// TIA Portal project "deneme3" (V14)

(* hardware
DEVICE "HMI_1"  KTP600 Basic color PN
   slot 0: "KTP600 Basic color PN"  KTP600 Basic color PN  6AV6 647-0AD11-3AX0  12.0.0.0
   slot 1: "HMI_RT_1"  KTP600 Basic color PN  6AV6 647-0AD11-3AX0  12.0.0.0
   slot 5: "HMI_1.IE_CP_1"  PROFINET Interface  12.0.0.0
      slot 1: "PROFINET Interface_1"  PROFINET Interface
         slot 1: "Port_1"  Port
DEVICE "S7300/ET200M station_1"  S7-300 station
   slot 0: "Rail_0"  Rail  6ES7 390-1***0-0AA0
   slot 2: "PLC_1"  CPU 315-2 PN/DP  6ES7 315-2EH13-0AB0  V2.6
      slot 1: "MPI/DP interface_1"  X1
      slot 2: "PROFINET interface_1"  PN-IO
         slot 1: "Port_1"  Port
*)

// ===== PLC "PLC_1"  CPU 315-2 PN/DP =====

VAR_GLOBAL   // PLC tag table "Default tag table"
   "start" AT %I0.0 : Bool;
   "Tag_2" AT %Q0.0 : Bool;
   "stop" AT %I0.1 : Bool;
END_VAR

DATA_BLOCK "barkod_database"   // DB1
{ S7_Optimized_Access := 'FALSE' }
VERSION : 0.1
   VAR
      kayitli_barkodlar : Array[0..99] of Struct
         barkod : Int;
      END_STRUCT;
      secili_barkod : Struct
         barkod : Int;
      END_STRUCT;
      barkod_kaydet : Bool;
      barkod_arttir : Bool;
      barkod_azalt : Bool;
      i : Int;
      barkod_oku : Bool;
      barkod_sil : Bool;
      bos_barkod : Struct
         barkod : Int;
      END_STRUCT;
   END_VAR
BEGIN
END_DATA_BLOCK

FUNCTION "fonksiyon_barkod" : Void   // FC1, SCL
{ S7_Optimized_Access := 'FALSE' }
VERSION : 0.1
BEGIN
   IF "barkod_database".barkod_kaydet THEN //BARKOD KAYDETME
       "barkod_database".kayitli_barkodlar["barkod_database".i] := "barkod_database".secili_barkod;
   END_IF;
   IF "barkod_database".barkod_oku THEN //BARKOD OKUMA
       "barkod_database".secili_barkod := "barkod_database".kayitli_barkodlar["barkod_database".i];
   END_IF;
   IF "barkod_database".barkod_sil THEN
       "barkod_database".kayitli_barkodlar["barkod_database".i] := "barkod_database".bos_barkod ;
   END_IF;
END_FUNCTION

ORGANIZATION_BLOCK "Main"   // OB1, LAD
TITLE = "Main Program Sweep (Cycle)"
{ S7_Optimized_Access := 'FALSE' }
VERSION : 0.1
   VAR_TEMP
      OB1_EV_CLASS : Byte;   // Bits 0-3 = 1 (Coming event), Bits 4-7 = 1 (Event class 1)
      OB1_SCAN_1 : Byte;   // 1 (Cold restart scan 1 of OB 1), 3 (Scan 2-n of OB 1)
      OB1_PRIORITY : Byte;   // Priority of OB Execution
      OB1_OB_NUMBR : Byte;   // 1 (Organization block 1, OB1)
      OB1_RESERVED_1 : Byte;   // Reserved for system
      OB1_RESERVED_2 : Byte;   // Reserved for system
      OB1_PREV_CYCLE : Int;   // Cycle time of previous OB1 scan (milliseconds)
      OB1_MIN_CYCLE : Int;   // Minimum cycle time of OB1 (milliseconds)
      OB1_MAX_CYCLE : Int;   // Maximum cycle time of OB1 (milliseconds)
      OB1_DATE_TIME : Date_And_Time;   // Date and time OB1 started
   END_VAR
BEGIN

REGION Network 1
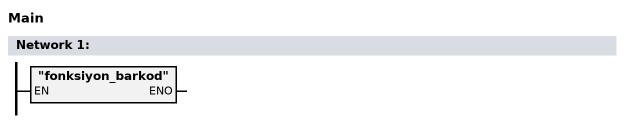
   RUNG wire#powerrail
      "fonksiyon_barkod"()
   END_RUNG
   // the same network as SCL:
   "fonksiyon_barkod"();
END_REGION
END_ORGANIZATION_BLOCK

(* ===== HMI "HMI_RT_1" =====
system functions are stored by id; their names below are inferred from use
connection "HMI_Connection_1": ETHERNET, SIMATIC S7 300/400 MPI

HMI tags "Default tag table"
   "barkod_database_secili_barkod.barkod" : Int = PLC barkod_database.secili_barkod.barkod AT %DB1.DBW200, 1 s
   "barkod_database_barkod_kaydet" : Bool = PLC barkod_database.barkod_kaydet AT %DB1.DBX202.0, 1 s
   "barkod_database_barkod_oku" : Bool = PLC barkod_database.barkod_oku AT %DB1.DBX206.0, 1 s
   "barkod_database_i" : Int = PLC barkod_database.i AT %DB1.DBW204, 1 s
   "barkod_database_barkod_sil" : Bool = PLC barkod_database.barkod_sil AT %DB1.DBX206.1, 1 s

Template "Template_1" 320x240
   Button "Exit" at 266,202 size 52x37; TextOff 'Exit'; PictureOff "ExitRuntime_KTP600_Basic_color_PN"; PictureOn "ExitRuntime_KTP600_Basic_color_PN"
      on Release: StopRuntime(0)
   Button "Template_Button" at 213,202 size 52x37; TextOff 'Text'
   Button "Template_Button_1" at 160,202 size 52x37; TextOff 'Text'
   Button "Template_Button_2" at 107,202 size 52x37; TextOff 'Text'
   Button "Template_Button_3" at 54,202 size 52x37; TextOff 'Text'
   Button "Start screen" at 1,202 size 52x37; TextOff 'Start screen'; PictureOff "NavigateHome_KTP600_Basic_color_PN"; PictureOn "NavigateHome_KTP600_Basic_color_PN"
      on Release: ActivateScreen("ilk sayfa", 0)

screen "ilk sayfa" 320x240, template "Template_1"
   TextField "HmiScreenItemData" at 32,3 size 256x17; Text 'Text'
   IOField "I/O field_1" at 150,3 size 111x35; FormatPattern s99999
      ProcessValue <- "barkod_database_secili_barkod.barkod"
   TextField "Text field_1" at 60,4 size 88x21; Text 'BARKOD :'
   Button "Button_1" at 37,129 size 105x36; TextOff 'BARKOD KAYDET'
      on Press: function_b14e0dd5("barkod_database_barkod_kaydet", 0)
   Button "Button_2" at 157,129 size 109x38; TextOff 'BARKOD OKU'
      on Press: function_b14e0dd5("barkod_database_barkod_oku", 0)
   Button "Button_3" at 168,81 size 96x32; TextOff 'Barkod no arrtır'
      on Press: function_dd21b452("barkod_database_i", 1); function_b14e0dd5("barkod_database_barkod_oku", 0)
   Button "Button_4" at 43,79 size 96x32; TextOff 'Barkod no azalt'
      on Press: function_b9b71300("barkod_database_i", 1); function_b14e0dd5("barkod_database_barkod_oku", 0)
   IOField "I/O field_2" at 157,51 size 96x23; FormatPattern s99999
      ProcessValue <- "barkod_database_i"
   TextField "Text field_2" at 70,48 size 72x15; Text 'BARKOD NO :'
   Button "Button_5" at 100,179 size 96x32; TextOff 'BARKOD SİL'
      on Press: function_b14e0dd5("barkod_database_barkod_sil", 0); function_b14e0dd5("barkod_database_barkod_oku", 0)
*)